Staubli VAL3: SpecialSeqVal.dtx

public num START_TRAJ_DOWN
public num START_TRAJ_STRE
public num END_TRAJECTORY
public num STOP_TRAJECTORY
